(* IEC 61131-3 sources: LabBench/Archive/Глобальные переменные, 5 files *)

(* ---- GVL_DiagSystem.st ---- *)
(*==============================================================================
    Название:    GVL_DiagSystem
    Автор:
    Дата:        2025-04-30
    Версия:      1.0

    Описание:    Глобальные переменные расширенной диагностической системы
==============================================================================*)
VAR_GLOBAL CONSTANT
    (* Количество ошибок и сценариев в системе *)
    MAX_ERRORS: UINT := 50;                  (* Максимальное количество ошибок *)
    MAX_SCENARIOS: UINT := 25;               (* Максимальное количество сценариев *)

    (* Идентификаторы систем *)
    SYSTEM_ID: WORD := 16#0100;              (* Общесистемные ошибки *)
    MEASUREMENT_ID: WORD := 16#0200;         (* Ошибки системы измерения *)
    EQUIPMENT_ID: WORD := 16#0300;           (* Ошибки оборудования *)
    COMMUNICATION_ID: WORD := 16#0400;       (* Ошибки связи *)

    (* Идентификаторы подсистем измерения *)
    PRESSURE_SENSORS_ID: WORD := 16#0210;    (* Датчики давления *)
    LEVEL_SENSORS_ID: WORD := 16#0220;       (* Датчики уровня *)
    FLOW_SENSORS_ID: WORD := 16#0230;        (* Расходомеры *)
    TEMP_SENSORS_ID: WORD := 16#0240;        (* Датчики температуры *)

    (* Идентификаторы оборудования *)
    PROP_VALVE_ID: WORD := 16#0310;          (* Пропорциональный клапан *)
    EM_VALVE_ID: WORD := 16#0320;            (* Электромагнитный клапан *)
    PUMP1_ID: WORD := 16#0330;               (* Насос 1 *)
    PUMP2_ID: WORD := 16#0340;               (* Насос 2 *)
    HEATER_ID: WORD := 16#0350;              (* Нагреватель (ТЭН) *)

    (* Идентификаторы связи *)
    SCADA_COMM_ID: WORD := 16#0410;          (* Связь со SCADA *)
    MODBUS_COMM_ID: WORD := 16#0420;         (* Связь по Modbus (ТРМ10) *)
END_VAR

VAR_GLOBAL
    (* Массивы ошибок и сценариев *)
    gaBlockingErrors: ARRAY[1..MAX_ERRORS] OF ST_BlockingError;     (* Массив ошибок *)
    gaDiagScenarios: ARRAY[1..MAX_SCENARIOS] OF ST_DiagScenario;    (* Массив сценариев *)

    (* Состояние системы *)
    geSystemState: E_SystemState;            (* Текущее состояние системы *)
    gxSystemBlockingRequired: BOOL;          (* Требуется блокировка системы *)
    gxSystemShutdownRequired: BOOL;          (* Требуется останов системы *)
    gxSystemResetRequired: BOOL;             (* Требуется сброс системы *)
    gstShutdownSequence: ST_ShutdownSequence;(* Последовательность останова *)

    (* Агрегированная информация о сценариях *)
    gxAnyScenarioActive: BOOL;               (* Любой сценарий активен *)
    gxAnyScenarioBlockingRequired: BOOL;     (* Любой сценарий требует блокировки *)
    gxAnyScenarioShutdownRequired: BOOL;     (* Любой сценарий требует останова *)
    gdwActiveScenariosMask: DWORD;           (* Битовая маска активных сценариев *)
    giLastActiveScenarioIndex: UINT;         (* Индекс последнего активного сценария *)

    (* Агрегированные состояния *)
    gxAnyError: BOOL;                        (* Флаг наличия любых ошибок *)
    gxSystemBlocking: BOOL;                  (* Флаг полной блокировки системы *)
    gdwActiveErrorMask: DWORD;               (* Битовая маска активных ошибок *)

    (* Блокировки устройств *)
    gxPropValveBlocking: BOOL;               (* Блокировка пропорционального клапана *)
    gxEMValveBlocking: BOOL;                 (* Блокировка электромагнитного клапана *)
    gxPump1Blocking: BOOL;                   (* Блокировка насоса 1 *)
    gxPump2Blocking: BOOL;                   (* Блокировка насоса 2 *)
    gxHeaterBlocking: BOOL;                  (* Блокировка нагревателя *)

    (* Управление лампой *)
    geLampMode: E_LampBlinkMode;             (* Режим работы сигнальной лампы *)
    gxLampState: BOOL;                       (* Текущее состояние лампы *)

    (* Команды управления *)
    gxResetAll: BOOL;                        (* Сброс всех ошибок *)
    gxResetMeasurement: BOOL;                (* Сброс ошибок измерительной системы *)
    gxResetPropValve: BOOL;                  (* Сброс ошибок пропорционального клапана *)
    gxResetEMValve: BOOL;                    (* Сброс ошибок электромагнитного клапана *)
    gxResetPump1: BOOL;                      (* Сброс ошибок насоса 1 *)
    gxResetPump2: BOOL;                      (* Сброс ошибок насоса 2 *)
    gxResetHeater: BOOL;                     (* Сброс ошибок нагревателя *)
    gxStartNormalShutdown: BOOL;             (* Запуск нормального останова *)
    gxStartEmergencyShutdown: BOOL;          (* Запуск аварийного останова *)
END_VAR

(* ---- GVL_Equipments.st ---- *)
(*==============================================================================
    Название:    GVL_Equipments
    Автор:       Редько А.
    Дата:        2025-04-27
    Версия:      1.0

    Описание:    Глобальные переменные оборудования
==============================================================================*)
VAR_GLOBAL
    (* Структуры данных оборудования *)
    stPropValve: ST_PropValve;       (* Пропорциональный кран *)
    stEMValve: ST_EMValve;            (* Электромагнитный клапан *)
END_VAR

(* ---- GVL_Inputs.st ---- *)
(*==============================================================================
    Название:    GVL_Inputs
    Автор:       Редько А.
    Дата:        2025-04-23
    Версия:      1.0

    Описание:    Глобальные переменные системы датчиков
==============================================================================*)
VAR_GLOBAL
    (* Датчики уровня *)
    GVL_stHydroLevel_KIE1: 		ST_HydroLevel_Data;     	(* Структура гидростатического датчика уровня в емкости КИЕ1 *)
    GVL_stFloatLevelSensors:    ST_FloatLevelGroup_Data;    (* Структура группы поплавковых датчиков уровня *)

    (* Датчики давления *)
    GVL_stPressureKIE2: 		ST_PressureSensor_Data;		(* Структура датчика давления в емкости КИЕ2 *)
    GVL_stPressurePipe: 		ST_PressureSensor_Data;   	(* Структура датчика давления в трубопроводе *)
    GVL_stPressurePumpIn1:		ST_PressureSensor_Data;  	(* Структура датчика давления перед насосом 1 *)
    GVL_stPressurePumpOut1:     ST_PressureSensor_Data;  	(* Структура датчика давления после насоса 1 *)
    GVL_stPressurePumpIn2: 		ST_PressureSensor_Data;  	(* Структура датчика давления перед насосом 2 *)
    GVL_stPressurePumpOut2: 	ST_PressureSensor_Data;  	(* Структура датчика давления после насоса 2 *)

    (* Датчики расхода *)
    GVL_stFlowSensor_PumpOut1: ST_FlowSensor_Data; (* Расходомер после насоса 1 *)
    GVL_stFlowSensor_PumpOut2: ST_FlowSensor_Data; (* Расходомер после насоса 2 *)
    GVL_stFlowSensor_Pipe: ST_FlowSensor_Data;     (* Расходомер в трубопроводе *)
END_VAR

(* ---- GVL_SCADA.st ---- *)
(*==============================================================================
    Название:    GVL_SCADA
    Автор:       Редько А.
    Дата:        2025-05-01
    Версия:      3.0

    Описание:    Глобальные переменные для интерфейса SCADA через OPC
                 - Оптимизированы типы данных для совместимости с OPC
                 - Используется явное управление режимами каждого устройства
                 - Heartbeat реализован как счетчик

                 Структура именования:
                 - GVL_SCADA_in_* : переменные только для записи (SCADA -> ПЛК)
                 - GVL_SCADA_out_* : переменные только для чтения (ПЛК -> SCADA)
                 - GVL_SCADA_inout_* : переменные для чтения и записи
==============================================================================*)
VAR_GLOBAL
    (* ======== СИСТЕМНЫЕ ПЕРЕМЕННЫЕ ======== *)
    (* Системные команды (SCADA -> ПЛК) *)
    GVL_SCADA_in_System_ResetAllErrors: BOOL := FALSE;     (* Общий сброс всех ошибок *)

    (* Системные статусы (ПЛК -> SCADA) *)
    GVL_SCADA_out_System_Heartbeat: DWORD;                (* Счетчик Heartbeat, циклически увеличивается *)
    GVL_SCADA_out_System_CycleTime_ms: DINT;              (* Время цикла в мс *)
    GVL_SCADA_out_System_ErrorCode: WORD;                 (* Код ошибки системы *)
    GVL_SCADA_out_System_ErrorCount: DWORD;               (* Счетчик ошибок *)

    (* ======== ПРОПОРЦИОНАЛЬНЫЙ КРАН ======== *)
    (* Команды управления (SCADA -> ПЛК) *)
    GVL_SCADA_in_PropValve_Mode: DINT := 1;               (* Режим работы: 0=AUTO, 1=MANUAL, 2=DISABLED, 3=E_STOP *)
    GVL_SCADA_in_PropValve_SetPosition: REAL := 0.0;      (* Задание положения (0-100%) *)
    GVL_SCADA_in_PropValve_Reset: BOOL := FALSE;          (* Сброс ошибок *)

    (* Настройки (SCADA -> ПЛК) *)
    GVL_SCADA_in_PropValve_SafePosition: REAL := 0.0;     (* Безопасное положение (0-100%) *)
    GVL_SCADA_in_PropValve_CloseThreshold: REAL := 2.0;   (* Порог "закрыт" (%) *)
    GVL_SCADA_in_PropValve_OpenThreshold: REAL := 98.0;   (* Порог "открыт" (%) *)
    GVL_SCADA_in_PropValve_Deadband: REAL := 1.0;         (* Зона нечувствительности (%) *)
    GVL_SCADA_in_PropValve_PositionTimeout_ms: DINT := 8000; (* Таймаут позиционирования в мс *)
    GVL_SCADA_in_PropValve_StuckTimeout_ms: DINT := 5000;    (* Таймаут заклинивания в мс *)

    (* Текущие значения (ПЛК -> SCADA) *)
    GVL_SCADA_out_PropValve_ActualPosition: REAL;         (* Текущее положение (0-100%) *)
    GVL_SCADA_out_PropValve_TargetPosition: REAL;         (* Целевое положение (0-100%) *)
    GVL_SCADA_out_PropValve_Mode: DINT;                   (* Текущий режим: 0=AUTO, 1=MANUAL, 2=DISABLED, 3=E_STOP *)
    GVL_SCADA_out_PropValve_State: DINT;                  (* Состояние: 0=CLOSED, 1=OPENING, 2=OPEN, 3=CLOSING,
                                                                         4=INTERMEDIATE, 5=REGULATING, 6=ERROR *)
    GVL_SCADA_out_PropValve_ErrorCode: WORD;              (* Код ошибки *)
    GVL_SCADA_out_PropValve_Valid: BOOL;                  (* Флаг достоверности данных *)
    GVL_SCADA_out_PropValve_Moving: BOOL;                 (* Флаг движения крана *)

    (* ======== ЭЛЕКТРОМАГНИТНЫЙ КЛАПАН ======== *)
    (* Команды управления (SCADA -> ПЛК) *)
    GVL_SCADA_in_EMValve_Mode: DINT := 1;                 (* Режим работы: 0=AUTO, 1=MANUAL, 2=DISABLED, 3=E_STOP *)
    GVL_SCADA_in_EMValve_Open: BOOL := FALSE;             (* Команда открытия в ручном режиме *)
    GVL_SCADA_in_EMValve_AutoOpen: BOOL := FALSE;         (* Команда от внешнего регулятора *)
    GVL_SCADA_in_EMValve_Reset: BOOL := FALSE;            (* Сброс счетчиков *)

    (* Настройки (SCADA -> ПЛК) *)
    GVL_SCADA_in_EMValve_WarningTime_ms: DINT := 900000;  (* Порог предупреждения в мс (15 мин) *)

    (* Текущие значения (ПЛК -> SCADA) *)
    GVL_SCADA_out_EMValve_IsOpen: BOOL;                   (* Текущее состояние *)
    GVL_SCADA_out_EMValve_Mode: DINT;                     (* Текущий режим: 0=AUTO, 1=MANUAL, 2=DISABLED, 3=E_STOP *)
    GVL_SCADA_out_EMValve_State: DINT;                    (* Состояние: 0=CLOSED, 1=OPEN, 2=LONG_OPERATION *)
    GVL_SCADA_out_EMValve_ContinuousOpTime_ms: DINT;      (* Время непрерывной работы в мс *)
    GVL_SCADA_out_EMValve_TotalOpTime_ms: DINT;           (* Общее время работы в мс *)
    GVL_SCADA_out_EMValve_WarningThreshold_ms: DINT;      (* Текущий порог предупреждения в мс *)

    (* ======== ДАТЧИКИ УРОВНЯ ======== *)
    (* Гидростатический датчик уровня КИЕ1 *)
    (* Настройки (SCADA -> ПЛК) *)
    GVL_SCADA_in_Level_KIE1_MaxLevelMM: REAL := 500.0;    (* Максимальный уровень, мм *)
    GVL_SCADA_in_Level_KIE1_Density: REAL := 1000.0;      (* Плотность жидкости, кг/м³ *)
    GVL_SCADA_in_Level_KIE1_LevelOffset: REAL := -1.0;    (* Смещение уровня, мм *)
    GVL_SCADA_in_Level_KIE1_Reset: BOOL := FALSE;         (* Сброс ошибок *)

    (* Текущие значения (ПЛК -> SCADA) *)
    GVL_SCADA_out_Level_KIE1_LevelMM: REAL;               (* Уровень в мм *)
    GVL_SCADA_out_Level_KIE1_LevelPercent: REAL;          (* Уровень в процентах *)
    GVL_SCADA_out_Level_KIE1_RawPressurePa: REAL;         (* Исходное давление в Па *)
    GVL_SCADA_out_Level_KIE1_Status: DINT;                (* Статус датчика *)
    GVL_SCADA_out_Level_KIE1_ErrorCode: WORD;             (* Код ошибки *)
    GVL_SCADA_out_Level_KIE1_Valid: BOOL;                 (* Достоверность данных *)

    (* Поплавковые датчики уровня *)
    (* Настройки (SCADA -> ПЛК) *)
    GVL_SCADA_in_FloatLevel_Reset: BOOL := FALSE;          (* Сброс ошибок *)

    (* Текущие значения (ПЛК -> SCADA) *)
    GVL_SCADA_out_FloatLevel_Low: BOOL;                   (* Состояние нижнего датчика *)
    GVL_SCADA_out_FloatLevel_Mid: BOOL;                   (* Состояние среднего датчика *)
    GVL_SCADA_out_FloatLevel_High: BOOL;                  (* Состояние верхнего датчика *)
    GVL_SCADA_out_FloatLevel_EstimationMM: REAL;          (* Оценка уровня в мм *)
    GVL_SCADA_out_FloatLevel_Percent: REAL;               (* Оценка уровня в процентах *)
    GVL_SCADA_out_FloatLevel_Status: DINT;                (* Статус датчиков *)
    GVL_SCADA_out_FloatLevel_ErrorCode: WORD;             (* Код ошибки *)
    GVL_SCADA_out_FloatLevel_Valid: BOOL;                 (* Достоверность данных *)

    (* ======== ДАТЧИКИ ДАВЛЕНИЯ ======== *)
    (* Общие настройки *)
    GVL_SCADA_in_Pressure_Reset: BOOL := FALSE;           (* Общий сброс ошибок датчиков давления *)

    (* Датчик в емкости КИЕ2 *)
    GVL_SCADA_in_Pressure_KIE2_MaxKPa: REAL := 200.0;     (* Максимальное давление, кПа *)
    GVL_SCADA_out_Pressure_KIE2_PressureKPa: REAL;        (* Давление в кПа *)
    GVL_SCADA_out_Pressure_KIE2_Status: DINT;             (* Статус датчика *)
    GVL_SCADA_out_Pressure_KIE2_ErrorCode: WORD;          (* Код ошибки *)
    GVL_SCADA_out_Pressure_KIE2_Valid: BOOL;              (* Достоверность данных *)

    (* Датчик в трубопроводе *)
    GVL_SCADA_in_Pressure_Pipe_MaxKPa: REAL := 300.0;     (* Максимальное давление, кПа *)
    GVL_SCADA_out_Pressure_Pipe_PressureKPa: REAL;        (* Давление в кПа *)
    GVL_SCADA_out_Pressure_Pipe_Status: DINT;             (* Статус датчика *)
    GVL_SCADA_out_Pressure_Pipe_ErrorCode: WORD;          (* Код ошибки *)
    GVL_SCADA_out_Pressure_Pipe_Valid: BOOL;              (* Достоверность данных *)

    (* Датчик перед насосом 1 *)
    GVL_SCADA_in_Pressure_PumpIn1_MaxKPa: REAL := 250.0;  (* Максимальное давление, кПа *)
    GVL_SCADA_out_Pressure_PumpIn1_PressureKPa: REAL;     (* Давление в кПа *)
    GVL_SCADA_out_Pressure_PumpIn1_Status: DINT;          (* Статус датчика *)
    GVL_SCADA_out_Pressure_PumpIn1_ErrorCode: WORD;       (* Код ошибки *)
    GVL_SCADA_out_Pressure_PumpIn1_Valid: BOOL;           (* Достоверность данных *)

    (* Датчик после насоса 1 *)
    GVL_SCADA_in_Pressure_PumpOut1_MaxKPa: REAL := 250.0; (* Максимальное давление, кПа *)
    GVL_SCADA_out_Pressure_PumpOut1_PressureKPa: REAL;    (* Давление в кПа *)
    GVL_SCADA_out_Pressure_PumpOut1_Status: DINT;         (* Статус датчика *)
    GVL_SCADA_out_Pressure_PumpOut1_ErrorCode: WORD;      (* Код ошибки *)
    GVL_SCADA_out_Pressure_PumpOut1_Valid: BOOL;          (* Достоверность данных *)

    (* Датчик перед насосом 2 *)
    GVL_SCADA_out_Pressure_PumpIn2_PressureKPa: REAL;     (* Давление в кПа *)
    GVL_SCADA_out_Pressure_PumpIn2_Status: DINT;          (* Статус датчика *)
    GVL_SCADA_out_Pressure_PumpIn2_ErrorCode: WORD;       (* Код ошибки *)
    GVL_SCADA_out_Pressure_PumpIn2_Valid: BOOL;           (* Достоверность данных *)

    (* Датчик после насоса 2 *)
    GVL_SCADA_out_Pressure_PumpOut2_PressureKPa: REAL;    (* Давление в кПа *)
    GVL_SCADA_out_Pressure_PumpOut2_Status: DINT;         (* Статус датчика *)
    GVL_SCADA_out_Pressure_PumpOut2_ErrorCode: WORD;      (* Код ошибки *)
    GVL_SCADA_out_Pressure_PumpOut2_Valid: BOOL;          (* Достоверность данных *)

    (* ======== РАСХОДОМЕРЫ ======== *)
    (* Общие настройки *)
    GVL_SCADA_in_Flow_Reset: BOOL := FALSE;               (* Общий сброс ошибок расходомеров *)

    (* Расходомер после насоса 1 *)
    GVL_SCADA_in_Flow_PumpOut1_Reset: BOOL := FALSE;      (* Сброс счетчика *)
    GVL_SCADA_out_Flow_PumpOut1_FlowLPM: REAL;            (* Расход в л/мин *)
    GVL_SCADA_out_Flow_PumpOut1_FlowM3H: REAL;            (* Расход в м³/ч *)
    GVL_SCADA_out_Flow_PumpOut1_TotalLiters: REAL;        (* Общий объем в литрах *)
    GVL_SCADA_out_Flow_PumpOut1_FrequencyHz: REAL;        (* Частота импульсов в Гц *)
    GVL_SCADA_out_Flow_PumpOut1_Status: DINT;             (* Статус датчика *)
    GVL_SCADA_out_Flow_PumpOut1_ErrorCode: WORD;          (* Код ошибки *)
    GVL_SCADA_out_Flow_PumpOut1_Valid: BOOL;              (* Достоверность данных *)

    (* Расходомер после насоса 2 *)
    GVL_SCADA_in_Flow_PumpOut2_Reset: BOOL := FALSE;      (* Сброс счетчика *)
    GVL_SCADA_out_Flow_PumpOut2_FlowLPM: REAL;            (* Расход в л/мин *)
    GVL_SCADA_out_Flow_PumpOut2_FlowM3H: REAL;            (* Расход в м³/ч *)
    GVL_SCADA_out_Flow_PumpOut2_TotalLiters: REAL;        (* Общий объем в литрах *)
    GVL_SCADA_out_Flow_PumpOut2_FrequencyHz: REAL;        (* Частота импульсов в Гц *)
    GVL_SCADA_out_Flow_PumpOut2_Status: DINT;             (* Статус датчика *)
    GVL_SCADA_out_Flow_PumpOut2_ErrorCode: WORD;          (* Код ошибки *)
    GVL_SCADA_out_Flow_PumpOut2_Valid: BOOL;              (* Достоверность данных *)

    (* Расходомер в трубопроводе *)
    GVL_SCADA_in_Flow_Pipe_Reset: BOOL := FALSE;          (* Сброс счетчика *)
    GVL_SCADA_out_Flow_Pipe_FlowLPM: REAL;                (* Расход в л/мин *)
    GVL_SCADA_out_Flow_Pipe_FlowM3H: REAL;                (* Расход в м³/ч *)
    GVL_SCADA_out_Flow_Pipe_TotalLiters: REAL;            (* Общий объем в литрах *)
    GVL_SCADA_out_Flow_Pipe_FrequencyHz: REAL;            (* Частота импульсов в Гц *)
    GVL_SCADA_out_Flow_Pipe_Status: DINT;                 (* Статус датчика *)
    GVL_SCADA_out_Flow_Pipe_ErrorCode: WORD;              (* Код ошибки *)
    GVL_SCADA_out_Flow_Pipe_Valid: BOOL;                  (* Достоверность данных *)
END_VAR

(* ---- GVL_SCADA_DiagSystem.st ---- *)
(*==============================================================================
    Название:    GVL_SCADA_DiagSystem
    Автор:
    Дата:        2025-04-28
    Версия:      1.0

    Описание:    Глобальные переменные для обмена данными со SCADA
                 по диагностике и блокировкам
==============================================================================*)
VAR_GLOBAL
    (* ======== КОМАНДЫ ОТ SCADA (SCADA -> ПЛК) ======== *)
    GVL_SCADA_in_Reset_All: BOOL := FALSE;           (* Общий сброс всех ошибок *)
    GVL_SCADA_in_Reset_Measurement: BOOL := FALSE;   (* Сброс ошибок измерительной системы *)
    GVL_SCADA_in_Reset_PropValve: BOOL := FALSE;     (* Сброс ошибок пропорционального клапана *)
    GVL_SCADA_in_Reset_EMValve: BOOL := FALSE;       (* Сброс ошибок электромагнитного клапана *)
    GVL_SCADA_in_Reset_Pump1: BOOL := FALSE;         (* Сброс ошибок насоса 1 *)
    GVL_SCADA_in_Reset_Pump2: BOOL := FALSE;         (* Сброс ошибок насоса 2 *)

    (* ======== ИНФОРМАЦИЯ ДЛЯ SCADA (ПЛК -> SCADA) ======== *)
    GVL_SCADA_out_AnyError: BOOL;                    (* Флаг наличия любых ошибок *)
    GVL_SCADA_out_SystemBlocking: BOOL;              (* Флаг полной блокировки системы *)
    GVL_SCADA_out_LampState: BOOL;                   (* Текущее состояние лампы *)
    GVL_SCADA_out_LampMode: DINT;                    (* Режим работы лампы *)
    GVL_SCADA_out_ErrorMask: DWORD;                  (* Битовая маска активных ошибок *)

    (* Состояния блокировок устройств *)
    GVL_SCADA_out_PropValveBlocking: BOOL;           (* Блокировка пропорционального клапана *)
    GVL_SCADA_out_EMValveBlocking: BOOL;             (* Блокировка электромагнитного клапана *)
    GVL_SCADA_out_Pump1Blocking: BOOL;               (* Блокировка насоса 1 *)
    GVL_SCADA_out_Pump2Blocking: BOOL;               (* Блокировка насоса 2 *)
END_VAR
